Staubli VAL3: robotStatusInq.pgx

public program robotStatusInq(num& x_nCyclePeriod[], tool& x_tExecuteTool[], frame& x_fRefFrame[], jointRx& x_jJointPos[], num& x_nJointVel[], num& x_nJointAccel[], pointRx& x_pPointPos[], num& x_nPointVel[], num& x_nPointAccel[], num& x_nResultantVel[], RobotMotionMsg& RobotMotion[])
  local num l_nNum
begin

  //This program is used for acquiring the current robot status which include joint space information(joint position,
  //joint velocity, joint acceleration) and cartesian space information(cartesian position, cartesian velocity, cartesian
  //acceleration). The current robot status are used for motion control and feedback information for host ROS controller.
  //According to last robot status based on specified frame and inqury period, the current joint positions, joint velocities,
  //cartesian positions and cartesian velocities of robot will be acquired and the current joint acceleration and cartesian
  //acceleration of robot will be calculated using differential method. The unit of the variables should be noticed extremely
  //in cartesian space and joint space.

  //Acquire the current status of robot from the encoders in joint space.(Unit: degree, degree/second, degree/(second squared))
  RobotMotion.jJointPos=$getJntFbk()
  $getJntSpeedFbk(x_nJointVel)
  //Calculate the joint acceleration of robot based on last robot status and inqury period.
  for l_nNum=0 to 5
    x_nJointAccel[l_nNum]=(x_nJointVel[l_nNum]-nNowJointVel[l_nNum])/x_nCyclePeriod
  endFor

  //Acquire the current status of robot from the encoders in cartesian space.(Unit: millimeter;degree, mm;°/s, mm;°/s^2)
  x_pPointPos=$getPosFbk(x_tExecuteTool,x_fRefFrame)
  x_nResultantVel=$getSpeedFbk(x_tExecuteTool,x_fRefFrame,x_nPointVel[0],x_nPointVel[1],x_nPointVel[2],x_nPointVel[3],x_nPointVel[4],x_nPointVel[5])
  for l_nNum=0 to 5
    x_nPointAccel[l_nNum]=(x_nPointVel[l_nNum]-nNowPointVel[l_nNum])/x_nCyclePeriod
  endFor


end
